Fanuc KAREL source: GN_CK_PNM_F9.KL

PROGRAM GN_CK_PNM_F9

%COMMENT = 'Check Parts vs Pallet Slots'
%NOLOCKGROUP
%NOPAUSE = ERROR + COMMAND + TPENABLE

%ENVIRONMENT REGOPE
%ENVIRONMENT STRNG
%ENVIRONMENT SYSDEF

CONST
   -- Input registers
   R_PLT_SLT = 427
   R_PRT_CNT = 404

   -- Status string register
   SR_STATUS = 44

VAR
   pallet_slots : INTEGER
   part_count   : INTEGER

   is_real      : BOOLEAN
   i_val        : INTEGER
   r_val        : REAL
   status       : INTEGER
   dummy        : INTEGER

BEGIN

   SET_STR_REG(SR_STATUS,'CHECKING PART COUNT',dummy)

   -- Read pallet slots
   GET_REG(R_PLT_SLT,is_real,i_val,r_val,status)

   IF status <> 0 THEN
      SET_STR_REG(SR_STATUS,'ERROR READING PALLET SLOTS',dummy)
      WRITE('ERROR READING R[427]',CR)
      RETURN
   ENDIF

   IF is_real THEN
      IF r_val <= 0 THEN
         SET_STR_REG(SR_STATUS,'INVALID PALLET SLOTS',dummy)
         RETURN
      ENDIF

      IF r_val <> TRUNC(r_val) THEN
         SET_STR_REG(SR_STATUS,'PALLET SLOTS NOT INTEGER',dummy)
         RETURN
      ENDIF

      pallet_slots = TRUNC(r_val)
   ELSE
      pallet_slots = i_val
   ENDIF

   IF pallet_slots <= 0 THEN
      SET_STR_REG(SR_STATUS,'INVALID PALLET SLOTS',dummy)
      RETURN
   ENDIF

   -- Read requested part count
   GET_REG(R_PRT_CNT,is_real,i_val,r_val,status)

   IF status <> 0 THEN
      SET_STR_REG(SR_STATUS,'ERROR READING PART COUNT',dummy)
      WRITE('ERROR READING R[404]',CR)
      RETURN
   ENDIF

   IF is_real THEN
      IF r_val <= 0 THEN
         SET_STR_REG(SR_STATUS,'INVALID PART COUNT',dummy)
         RETURN
      ENDIF

      IF r_val <> TRUNC(r_val) THEN
         SET_STR_REG(SR_STATUS,'PART COUNT NOT INTEGER',dummy)
         RETURN
      ENDIF

      part_count = TRUNC(r_val)
   ELSE
      part_count = i_val
   ENDIF

   IF part_count <= 0 THEN
      SET_STR_REG(SR_STATUS,'INVALID PART COUNT',dummy)
      RETURN
   ENDIF

   -- Compare part count against pallet capacity
   IF part_count <= pallet_slots THEN
      SET_STR_REG(SR_STATUS,'OK',dummy)
      WRITE('NUMBER OF PARTS IS OK',CR)
   ELSE
      SET_STR_REG(SR_STATUS,'PART COUNT EXCEEDS SLOTS',dummy)
      WRITE('PART COUNT EXCEEDS PALLET SLOTS',CR)
   ENDIF

END GN_CK_PNM_F9
